(* PLC project cmd_agitator_1speed, Dassault Systèmes ControlBuild 2024x *)
(* stored: creationDateTime 2023-10-03T11:13:36-01:00 *)

FUNCTION_BLOCK actuator
  VAR_INPUT
    autoMode : BOOL := false;
    manualMode : BOOL := false;
  END_VAR
  VAR_INPUT
    autoCmd : BOOL := false;
  END_VAR
  VAR_INPUT
    forwardPB : BOOL := false;
    stopPB : BOOL := false;
  END_VAR
  VAR_INPUT
    generalFault : BOOL := false;
  END_VAR
  VAR_OUTPUT
    cmd : BOOL := false;
  END_VAR

(* LD diagram, written out as Structured Text *)
1:
cmd := (autoMode AND autoCmd OR manualMode AND (forwardPB OR cmd) AND NOT stopPB) AND NOT generalFault;
END_FUNCTION_BLOCK

FUNCTION_BLOCK faults
  VAR_INPUT
    cmd : BOOL := false;
  END_VAR
  VAR_INPUT
    thermalFB : BOOL := false;
    cmdFB : BOOL := false;
  END_VAR
  VAR_INPUT
    acknowledgePB : BOOL := false;
  END_VAR
  VAR_OUTPUT
    generalFault : BOOL := false;
  END_VAR
  VAR
    thermalFault : BOOL := false;
    cmdFBFault : BOOL := false;
  END_VAR

(* LD diagram, written out as Structured Text *)
1:
IF acknowledgePB THEN thermalFault := FALSE; END_IF;
IF acknowledgePB THEN cmdFBFault := FALSE; END_IF;
IF acknowledgePB THEN generalFault := FALSE; END_IF;
2:
TON_FB(IN := cmd, PT := T#0h0m2s0ms);
IF TON_FB.Q0 AND NOT cmdFB THEN cmdFBFault := TRUE; END_IF;
3:
IF NOT thermalFB THEN thermalFault := TRUE; END_IF;
4:
IF thermalFault OR cmdFBFault THEN generalFault := TRUE; END_IF;
END_FUNCTION_BLOCK

(* Command of a 1-speed motorized agitator with fault detection. *)
PROGRAM cmd_equipment_library.cmd_agitator_1speed
  VAR_INPUT
    autoMode : BOOL := false;
    manualMode : BOOL := false;
  END_VAR
  VAR_INPUT
    autoCmd : BOOL := false;
  END_VAR
  VAR_INPUT
    thermalFB : BOOL := false;
    cmdFB : BOOL := false;
  END_VAR
  VAR_INPUT
    forwardPB : BOOL := false;
    stopPB : BOOL := false;
  END_VAR
  VAR_INPUT
    acknowledgePB : BOOL := false;
  END_VAR
  VAR_OUTPUT
    cmd : BOOL := false;
  END_VAR
  VAR_OUTPUT
    generalFault : BOOL := false;
  END_VAR

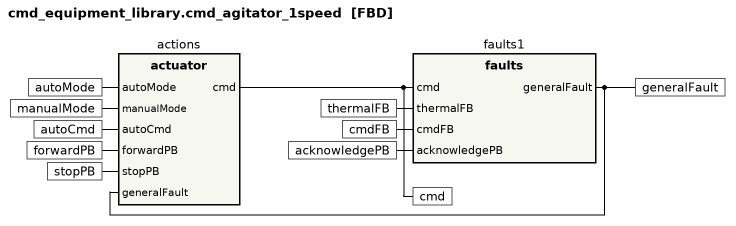
(* FBD diagram, written out as Structured Text *)
faults1(cmd := actions.cmd, thermalFB := thermalFB, cmdFB := cmdFB, acknowledgePB := acknowledgePB);
actions(autoMode := autoMode, manualMode := manualMode, autoCmd := autoCmd, forwardPB := forwardPB, stopPB := stopPB, generalFault := faults1.generalFault);
cmd := actions.cmd;
generalFault := faults1.generalFault;
END_PROGRAM
